{attribute 'linkalways'} 
{attribute 'no_explicit_call' := 'This FB is a CLASS and must be accessed using methods or properties'}
{attribute 'enable_dynamic_creation'}
FUNCTION_BLOCK _ETcVnCalibrationPattern EXTENDS EnumDatatypeBase
VAR
	localData : ETcVnCalibrationPattern;
	activeData : REFERENCE TO ETcVnCalibrationPattern;
	enumBaseDatatype : _DINT(localData);
END_VAR

METHOD PRIVATE AddLocalEnumeration
VAR_INPUT
	Enumeration : T_MAXSTRING;
	Value : ETcVnCalibrationPattern;
END_VAR
AddEnumeration(Enumeration, Value);
END_METHOD

PROPERTY PUBLIC Address : PVOID
GET
Address := ADR(activeData);
END_GET
END_PROPERTY

METHOD PUBLIC ClearReference
VAR_INPUT
END_VAR
activeData REF= localData;
SetBaseDatatypeReference();
END_METHOD

METHOD PUBLIC Clone : I_Datatype
VAR
    pClone : POINTER TO _ETcVnCalibrationPattern;
END_VAR
pClone := __NEW(_ETcVnCalibrationPattern(InitialValue := Value));
Clone := pClone^;
END_METHOD

METHOD FB_init : BOOL
VAR_INPUT
	bInitRetains : BOOL; // if TRUE, the retain variables are initialized (warm start / cold start)
	bInCopyCode : BOOL;  // if TRUE, the instance afterwards gets moved into the copy code (online change)
	InitialValue : ETcVnCalibrationPattern;
END_VAR
localData := InitialValue;
AddBaseDatatype(enumBaseDatatype);
ClearReference();

AddLocalEnumeration('TCVN_CP_CIRCLES_SYM', ETcVnCalibrationPattern.TCVN_CP_CIRCLES_SYM);
AddLocalEnumeration('TCVN_CP_CIRCLES_ASYM', ETcVnCalibrationPattern.TCVN_CP_CIRCLES_ASYM);
AddLocalEnumeration('TCVN_CP_CIRCLES_ASYM_INDENT', ETcVnCalibrationPattern.TCVN_CP_CIRCLES_ASYM_INDENT);
END_METHOD

PROPERTY PUBLIC Identifier : T_MAXSTRING
GET
Identifier := 'ETcVnCalibrationPattern';
END_GET
END_PROPERTY

METHOD IsEnumeratorValueEqual : BOOL
VAR_INPUT
	Enumerator : I_KeyValueForwardEnumerator;
END_VAR
VAR
	storedValue : ETcVnCalibrationPattern;
END_VAR
IF NOT Enumerator.TryGet(storedValue) THEN
	RETURN;
END_IF

IsEnumeratorValueEqual := storedValue = activeData;
END_METHOD

METHOD PUBLIC MakeReferenceTo
VAR_INPUT
	ReferenceTarget : REFERENCE TO ETcVnCalibrationPattern;
END_VAR
activeData REF= ReferenceTarget;
SetBaseDatatypeReference();
END_METHOD

METHOD PROTECTED SetBaseDatatypeReference
VAR_INPUT
END_VAR
enumBaseDatatype.MakeReferenceTo(activeData);
END_METHOD

PROPERTY PUBLIC Size : UDINT
GET
Size := SIZEOF(activeData);
END_GET
END_PROPERTY

METHOD TryMakeReferenceTo : BOOL
VAR_INPUT
	Target : I_Datatype;
END_VAR
VAR
	targetAsEnum : I_EnumDatatype;
	pTargetData : POINTER TO ETcVnCalibrationPattern;
END_VAR
IF NOT Target.TryResolveAsEnumDatatype(targetAsEnum) THEN
	RETURN;
END_IF

IF targetAsEnum.Identifier <> Identifier THEN
	RETURN;
END_IF

pTargetData := Target.Address;
activeData REF= pTargetData^;
SetBaseDatatypeReference();
TryMakeReferenceTo := TRUE;
END_METHOD

PROPERTY PUBLIC Value : ETcVnCalibrationPattern
GET
Value := activeData;
END_GET
SET
activeData := Value;
END_SET
END_PROPERTY

END_FUNCTION_BLOCK

(* stored: Version 1.1.0.1, ProductVersion 3.1.4024.12
   POU _ETcVnCalibrationPattern: Id {242b7478-690d-4c28-ab58-0771f86f04d1}, SpecialFunc None
   Folder Constructor: Id {052bf58e-5e75-4250-8666-3b9d80163253}
   Folder Private: Id {96d89ac4-5ec6-4c6f-b6d5-705b3acea75e}
   Folder Protected: Id {c95cf233-58df-454c-b43f-f514fde668b9}
   Method AddLocalEnumeration: Id {27784235-ed37-44c2-ad52-aef4feaedbb7}
   Property Address: Id {9938c10e-2f41-4128-b019-0de24ea63e5d}
   Get Get: Id {280976cc-1b1a-4bfd-940f-df086277eee9}
   Method ClearReference: Id {97e1dfc4-12aa-44ad-873e-b4a352aedbc3}
   Method Clone: Id {b06a644d-f512-402b-9c78-fa94ca876d2a}
   Method FB_init: Id {41dea6d3-5ac5-4887-8e07-4c2e9d3d334f}
   Property Identifier: Id {cf6ce56b-f9fb-4e8f-bcf4-45eb1baf4ca7}
   Get Get: Id {d637b286-1d02-4673-8d31-208312ec9c14}
   Method IsEnumeratorValueEqual: Id {36c49053-c56a-4947-8417-32197656628f}
   Method MakeReferenceTo: Id {f5071b5c-f603-42b4-a27f-6f4ff65c1844}
   Method SetBaseDatatypeReference: Id {638067ea-020c-41ad-b83e-4ab3ecf50f8c}
   Property Size: Id {4fe4ebf5-99ef-4cf0-854b-3ecc634d0735}
   Get Get: Id {5f609d7b-9fb1-461a-89f9-0d3a56508c19}
   Method TryMakeReferenceTo: Id {8ffa0e03-761f-4b19-ad58-7d91491f4e7a}
   Property Value: Id {92425e6b-21c4-400a-892f-54440ae8e267}
   Get Get: Id {bde5f00d-11c9-4d97-894e-2e46c53f46aa}
   Set Set: Id {f7a59fbb-830e-419d-b216-30ba25e1009f} *)
